# EPICS alarm handler configuration: apps/alhConfig/HPS.alhConfig
#===============================================================================
# HPS Top-level Alarm Config
#===============================================================================

GROUP    NULL                         HPS

$GUIDANCE
    For info on target-related items, please contact HPS Experts
$END

#=======================================
# Subsystems
#=======================================

INCLUDE HPS /usr/clas12/hps/prod/apps/alhConfig/beam.alhConfig
INCLUDE HPS /usr/clas12/hps/prod/apps/alhConfig/trigger.alhConfig
INCLUDE HPS /usr/clas12/hps/prod/apps/alhConfig/ecal.alhConfig
INCLUDE HPS /usr/clas12/hps/prod/apps/alhConfig/svt.alhConfig
INCLUDE HPS /usr/clas12/hps/prod/apps/alhConfig/hodo.alhConfig
INCLUDE HPS /usr/clas12/hps/prod/apps/alhConfig/magnets.alhConfig
INLCUDE HPS /usr/clas12/hps/prod/apps/alhConfig/iocs.alhConfig
